PROGRAM MAIN
VAR
		PushButton01			:	BOOL;
		PushButton02			:	BOOL;
		PushButton03			:	BOOL;
		Reset					:	BOOL;
		
		Buzzer					:	BOOL;
		Player01Light			:	BOOL;
		Player02Light			:	BOOL;
		Player03Light			:	BOOL;
		ton01					: 	TON;
END_VAR
VAR // added by the converter: edge detectors and wires of the graphical bodies
    _w1 : BOOL;
END_VAR

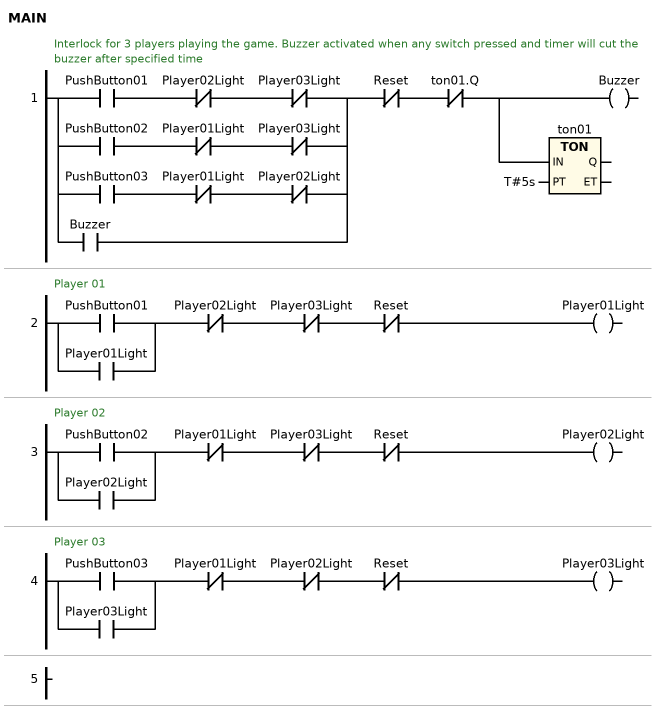
// NETWORK 1
// Interlock for 3 players playing the game. Buzzer activated when any switch pressed and timer will cut the buzzer after specified time
_w1 := (PushButton01 AND NOT Player02Light AND NOT Player03Light OR PushButton02 AND NOT Player01Light AND NOT Player03Light OR PushButton03 AND NOT Player01Light AND NOT Player02Light OR Buzzer) AND NOT Reset AND NOT ton01.Q;
Buzzer := _w1;
ton01(IN := _w1, PT := T#5s); // TON

// NETWORK 2
// Player 01
Player01Light := (PushButton01 OR Player01Light) AND NOT Player02Light AND NOT Player03Light AND NOT Reset;

// NETWORK 3
// Player 02
Player02Light := (PushButton02 OR Player02Light) AND NOT Player01Light AND NOT Player03Light AND NOT Reset;

// NETWORK 4
// Player 03
Player03Light := (PushButton03 OR Player03Light) AND NOT Player01Light AND NOT Player02Light AND NOT Reset;

// NETWORK 5

END_PROGRAM

(* stored: Version 1.1.0.1, ProductVersion 3.1.4024.15
   POU MAIN: Id {9b0b0180-3053-4bc5-9e1d-fd0445ae22a4}, SpecialFunc None *)
